(* IEC 61131-3 sources: eCockpitGit/test_project/src/%F%00 Library/%F%Common Functions/%F%String/%F%Normal/%F%Padd, 4 files *)

(* ---- %POU%FU_sPaddBack.st ---- *)
//This function padds the back of a string with the given character, the given amount
//If the padd amount plus the string is longer than the output string, the input string will be cut off to make space for the padding
// +-----------+----------+----------+-----------------------------------------------------------------------------------------------------------------------+
// |**Version**|**Author**| **Date** |**Changes**                                                                                                            |
// +-----------+----------+----------+-----------------------------------------------------------------------------------------------------------------------+
// | 1         | NSN      | 04-02-19 | Creation                                                                                                              |
// +-----------+----------+----------+-----------------------------------------------------------------------------------------------------------------------+
FUNCTION FU_sPaddBack : STRING(255)
VAR_INPUT
	sStr		:STRING(255);		//Input String
	wPadds		:WORD;				//How much to padd it
	eChar		:EASCII;		//Which character to padd with
END_VAR

(*%!%__DELIMITER__%!%*)
FU_sPaddBackBIBO(sOut:=FU_sPaddBack,sStr:=sStr,wPadds:=wPadds,wOutSize:=255,eChar:=eChar);

(* ---- %POU%FU_sPaddBackLen.st ---- *)
//This function padds the back of a string with the given character, the given amount
//If the padd amount plus the string is longer than the output string, the input string will be cut off to make space for the padding
// +-----------+----------+----------+-----------------------------------------------------------------------------------------------------------------------+
// |**Version**|**Author**| **Date** |**Changes**                                                                                                            |
// +-----------+----------+----------+-----------------------------------------------------------------------------------------------------------------------+
// | 1         | NSN      | 04-02-19 | Creation                                                                                                              |
// +-----------+----------+----------+-----------------------------------------------------------------------------------------------------------------------+
FUNCTION FU_sPaddBackLen  : STRING(255)
VAR_INPUT
	sStr		:STRING(255);		//Input String
	wLen		:WORD;				//How much to padd it
	eChar		:EASCII;		//Which character to padd with
END_VAR
(*%!%__DELIMITER__%!%*)
FU_sPaddBackLenBIBO(sOut:=FU_sPaddBackLen,sStr:=sStr,wLen:=wLen,wOutSize:=255,eChar:=eChar);

(* ---- %POU%FU_sPaddFront.st ---- *)
//This function padds the front of a string with the given character, the given amount
//If the padd amount plus the string is longer than the output string, the input string will be cut off to make space for the padding
// +-----------+----------+----------+-----------------------------------------------------------------------------------------------------------------------+
// |**Version**|**Author**| **Date** |**Changes**                                                                                                            |
// +-----------+----------+----------+-----------------------------------------------------------------------------------------------------------------------+
// | 1         | NSN      | 04-02-19 | Creation                                                                                                              |
// +-----------+----------+----------+-----------------------------------------------------------------------------------------------------------------------+
FUNCTION FU_sPaddFront : STRING(255)
VAR_INPUT
	sStr		:STRING(255);		//Input String
	wPadds		:WORD;				//How much to padd it
	eChar		:EASCII;		//Which character to padd with
END_VAR
(*%!%__DELIMITER__%!%*)
FU_sPaddFrontBIBO(sOut:=FU_sPaddFront,sStr:=sStr,wPadds:=wPadds,wOutSize:=255,eChar:=eChar);

(* ---- %POU%FU_sPaddFrontLen.st ---- *)
//This function padds the front of a string with the given character, the given amount
//If the padd amount plus the string is longer than the output string, the input string will be cut off to make space for the padding
// +-----------+----------+----------+-----------------------------------------------------------------------------------------------------------------------+
// |**Version**|**Author**| **Date** |**Changes**                                                                                                            |
// +-----------+----------+----------+-----------------------------------------------------------------------------------------------------------------------+
// | 1         | NSN      | 04-02-19 | Creation                                                                                                              |
// +-----------+----------+----------+-----------------------------------------------------------------------------------------------------------------------+
FUNCTION FU_sPaddFrontLen : STRING(255)
VAR_INPUT
	sStr		:STRING(255);		//Input String
	wLen		:WORD;				//How much to padd it
	eChar		:EASCII;		//Which character to padd with
END_VAR
(*%!%__DELIMITER__%!%*)
FU_sPaddFrontLenBIBO(sOut:=FU_sPaddFrontLen,sStr:=sStr,wLen:=wLen,wOutSize:=255,eChar:=eChar);
